Staubli VAL3: onF4Event.pgx

program onF4Event(bool& x_bSave[])
begin
  // look if the bButton is enable
  if bButton[3]
    // paste the items select
    call prog:pasteItem(nIndex)
    logMsg("[KERNEL] INTERFACE:Paste progs items")
    call buildList()
    x_bSave=true
  endIf
end
